// TIA Portal V16 export
// export: Created 2023-09-25T11:31:54.6330988Z, ExportSetting WithDefaults, DisplayName Totally Integrated Automation Portal, DisplayVersion V16 Update 6, DisplayName TIA Portal Version Control Interface, DisplayVersion V16 Update 2, DisplayName TIA Portal Openness, DisplayVersion V16 Update 6, DisplayName STEP 7 Professional, DisplayVersion V16 Update 6, DisplayName STEP 7 Safety, DisplayVersion V16, DisplayName WinCC Advanced, DisplayVersion V16 Update 6
DATA_BLOCK "ValueHz_in_Alarm_CurrentOver_DB"   // DB71
AUTHOR : rtecmer
VERSION : 0.1
// stored: AutoNumber true, DBAccessibleFromOPCUA true, InstanceOfName 06_M_Control Hz safe mode from bar Max, InstanceOfType FB
"06_M_Control Hz safe mode from bar Max"
   // VAR_INPUT
   //    Value_Max : Bool;
   //    My_1Hz : Bool;
   //    Act_Hz : Real;
   //    IsMotor2Set : Bool;
   //    IsMotor3Set : Bool;
   //    IsMotor4Set : Bool;
   //    IsReadyinverter1 : Bool;
   // END_VAR
   // VAR_OUTPUT
   //    Value_Manual_Hz : Real;
   //    Rst_Motor2 : Bool;
   //    Rst_Motor3 : Bool;
   //    Rst_Motor4 : Bool;
   //    Rst_Driver : Bool;
   // END_VAR
   // VAR
   //    set_NewValue { ExternalAccessible := 'False'; ExternalVisible := 'False'; ExternalWritable := 'False'} : Bool;
   //    index { ExternalAccessible := 'False'; ExternalVisible := 'False'; ExternalWritable := 'False'} : Bool;
   //    CV { ExternalAccessible := 'False'; ExternalVisible := 'False'; ExternalWritable := 'False'} : Int;
   //    load_cunt { ExternalAccessible := 'False'; ExternalVisible := 'False'; ExternalWritable := 'False'} : Bool;
   //    tmp_Hz { ExternalAccessible := 'False'; ExternalVisible := 'False'; ExternalWritable := 'False'} : Real;
   //    cnt_Hz { ExternalAccessible := 'False'; ExternalVisible := 'False'; ExternalWritable := 'False'} : Real;
   //    mem_Triger_Alarm { ExternalAccessible := 'False'; ExternalVisible := 'False'; ExternalWritable := 'False'} : Bool;
   // END_VAR
BEGIN
END_DATA_BLOCK
